// TIA Portal V19 export
FUNCTION "DATE & TIME FC" : Void   // FC9, LAD
{ S7_Optimized_Access := 'TRUE' }
// stored: SetENOAutomatically false
BEGIN

REGION Network 1
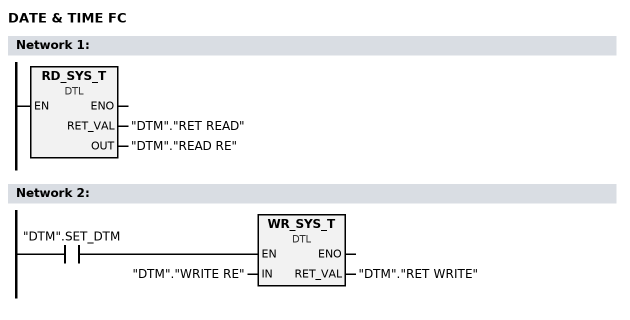
   RUNG wire#powerrail
      { S7_Templates := "date_type := DTL" } RD_SYS_T(RET_VAL => "DTM"."RET READ", OUT => "DTM"."READ RE")
   END_RUNG
   // the same network as SCL:
   "DTM"."RET READ" := RD_SYS_T(OUT => "DTM"."READ RE");
END_REGION

REGION Network 2
   RUNG wire#powerrail
      Contact( "DTM".SET_DTM )
      { S7_Templates := "date_type := DTL" } WR_SYS_T(IN := "DTM"."WRITE RE", RET_VAL => "DTM"."RET WRITE")
   END_RUNG
   // the same network as SCL:
   IF "DTM".SET_DTM THEN "DTM"."RET WRITE" := WR_SYS_T(IN := "DTM"."WRITE RE"); END_IF;
END_REGION
END_FUNCTION
